// TIA Portal project "SIMULACION" (V16)

(* hardware
DEVICE "S7-1200 station_1"  S7-1200 Station
   slot 0: "Rack_0"  S7-1200 Rack  Rack  V1.0
   slot 1: "PLC_1"  CPU 1214C DC/DC/Rly  6ES7 214-1HG40-0XB0  V4.0
*)

// ===== PLC "PLC_1"  CPU 1214C DC/DC/Rly =====

VAR_GLOBAL   // PLC tag table "Default tag table"
   "ET0" AT %M0.0 : Bool;
   "ET1" AT %M0.1 : Bool;
   "ET2" AT %M0.2 : Bool;
   "ET3" AT %M0.3 : Bool;
   "ET4" AT %M0.4 : Bool;
   "ET5" AT %M0.5 : Bool;
   "ET6" AT %M0.6 : Bool;
   "ET7" AT %M0.7 : Bool;
   "ET8" AT %M1.0 : Bool;
   "ET9" AT %M1.1 : Bool;
   "ET10" AT %M1.2 : Bool;
   "ET11" AT %M1.3 : Bool;
   "ET12" AT %M1.4 : Bool;
   "ET13" AT %M1.5 : Bool;
   "ET14" AT %M1.6 : Bool;
   "ET15" AT %M1.7 : Bool;
   "ET16" AT %M2.0 : Bool;
   "ET17" AT %M2.1 : Bool;
   "ET18" AT %M2.2 : Bool;
   "MARCHA" AT %I0.0 : Bool;
   "TANQUEA" AT %Q0.0 : Bool;
   "TANQUEB" AT %Q0.1 : Bool;
   "W1" AT %Q0.2 : Bool;
   "W2" AT %Q0.3 : Bool;
   "W3" AT %Q0.4 : Bool;
   "W4" AT %Q0.5 : Bool;
   "W5" AT %Q0.6 : Bool;
END_VAR

// folder: System blocks/Program resources

DATA_BLOCK "TW1"   // DB2
{ S7_Optimized_Access := 'TRUE' }
AUTHOR : Simatic
FAMILY : IEC
NAME : IEC_TMR
VERSION : 1.0
// stored: InstanceOfName IEC_TIMER
"IEC_TIMER"
BEGIN
END_DATA_BLOCK

DATA_BLOCK "TW2"   // DB3
{ S7_Optimized_Access := 'TRUE' }
AUTHOR : Simatic
FAMILY : IEC
NAME : IEC_TMR
VERSION : 1.0
// stored: InstanceOfName IEC_TIMER
"IEC_TIMER"
BEGIN
END_DATA_BLOCK

DATA_BLOCK "TW3"   // DB4
{ S7_Optimized_Access := 'TRUE' }
AUTHOR : Simatic
FAMILY : IEC
NAME : IEC_TMR
VERSION : 1.0
// stored: InstanceOfName IEC_TIMER
"IEC_TIMER"
BEGIN
END_DATA_BLOCK

DATA_BLOCK "T4"   // DB5
{ S7_Optimized_Access := 'TRUE' }
AUTHOR : Simatic
FAMILY : IEC
NAME : IEC_TMR
VERSION : 1.0
// stored: InstanceOfName IEC_TIMER
"IEC_TIMER"
BEGIN
END_DATA_BLOCK

DATA_BLOCK "T5"   // DB6
{ S7_Optimized_Access := 'TRUE' }
AUTHOR : Simatic
FAMILY : IEC
NAME : IEC_TMR
VERSION : 1.0
// stored: InstanceOfName IEC_TIMER
"IEC_TIMER"
BEGIN
END_DATA_BLOCK

DATA_BLOCK "T6"   // DB7
{ S7_Optimized_Access := 'TRUE' }
AUTHOR : Simatic
FAMILY : IEC
NAME : IEC_TMR
VERSION : 1.0
// stored: InstanceOfName IEC_TIMER
"IEC_TIMER"
BEGIN
END_DATA_BLOCK

DATA_BLOCK "T7"   // DB8
{ S7_Optimized_Access := 'TRUE' }
AUTHOR : Simatic
FAMILY : IEC
NAME : IEC_TMR
VERSION : 1.0
// stored: InstanceOfName IEC_TIMER
"IEC_TIMER"
BEGIN
END_DATA_BLOCK

DATA_BLOCK "T8"   // DB9
{ S7_Optimized_Access := 'TRUE' }
AUTHOR : Simatic
FAMILY : IEC
NAME : IEC_TMR
VERSION : 1.0
// stored: InstanceOfName IEC_TIMER
"IEC_TIMER"
BEGIN
END_DATA_BLOCK

// folder: (top level)

ORGANIZATION_BLOCK "Main"   // OB1, LAD, ProgramCycle
TITLE = "Main Program Sweep (Cycle)"
{ S7_Optimized_Access := 'TRUE' }
VERSION : 0.1
BEGIN

REGION Network 1: Estado Inicial
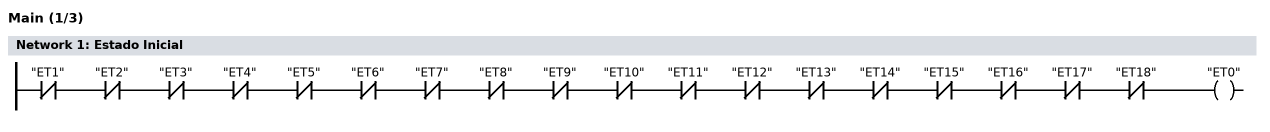
   RUNG wire#powerrail
      I_Contact( "ET1" )
      I_Contact( "ET2" )
      I_Contact( "ET3" )
      I_Contact( "ET4" )
      I_Contact( "ET5" )
      I_Contact( "ET6" )
      I_Contact( "ET7" )
      I_Contact( "ET8" )
      I_Contact( "ET9" )
      I_Contact( "ET10" )
      I_Contact( "ET11" )
      I_Contact( "ET12" )
      I_Contact( "ET13" )
      I_Contact( "ET14" )
      I_Contact( "ET15" )
      I_Contact( "ET16" )
      I_Contact( "ET17" )
      I_Contact( "ET18" )
      Coil( "ET0" )
   END_RUNG
   // the same network as SCL:
   "ET0" := NOT "ET1" AND NOT "ET2" AND NOT "ET3" AND NOT "ET4" AND NOT "ET5" AND NOT "ET6" AND NOT "ET7" AND NOT "ET8" AND NOT "ET9" AND NOT "ET10" AND NOT "ET11" AND NOT "ET12" AND NOT "ET13" AND NOT "ET14" AND NOT "ET15" AND NOT "ET16" AND NOT "ET17" AND NOT "ET18";
END_REGION

REGION Network 2: Etapas de transicion
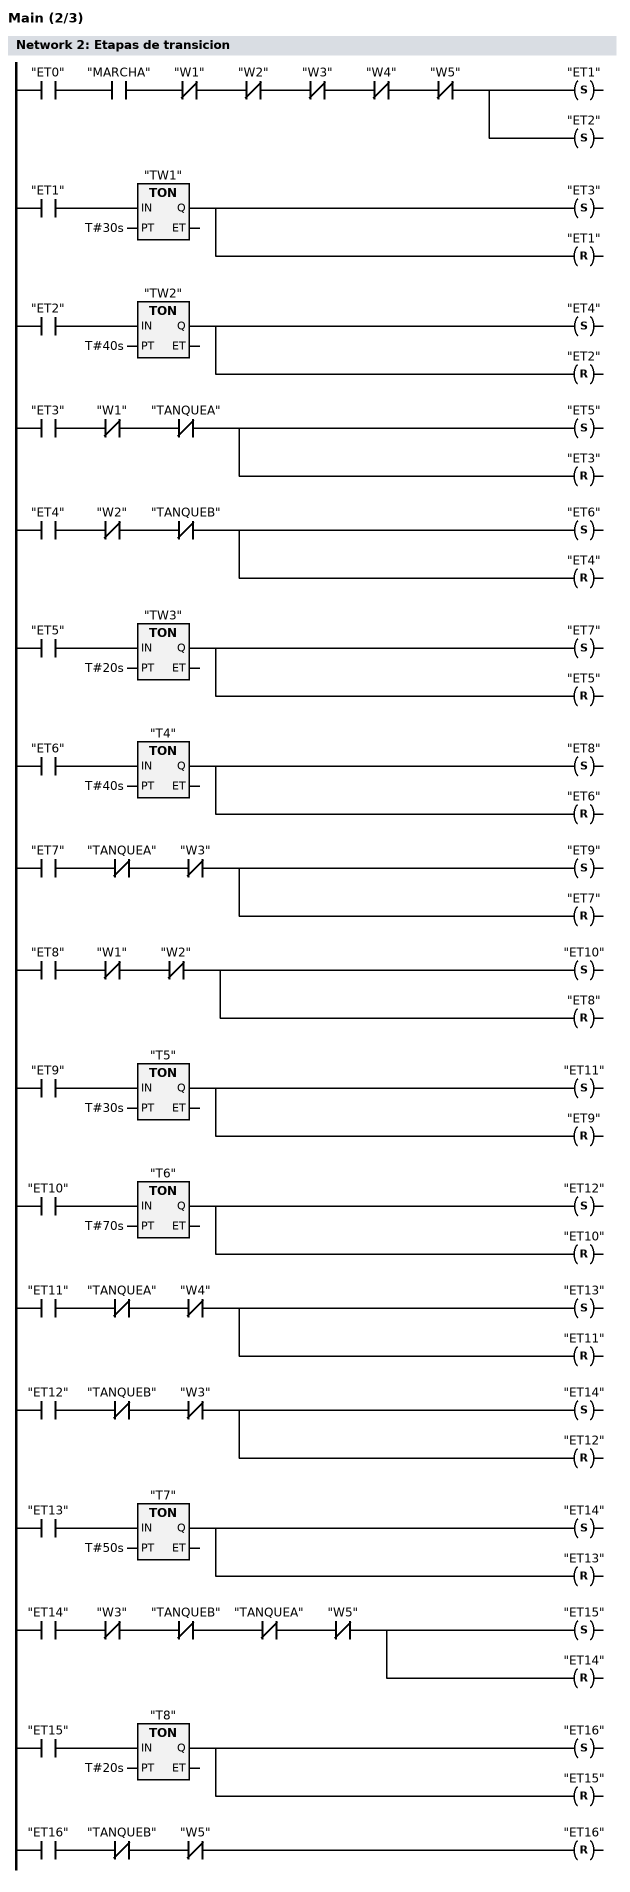
   IF "ET0" AND "MARCHA" AND NOT "W1" AND NOT "W2" AND NOT "W3" AND NOT "W4" AND NOT "W5" THEN
       "ET1" := TRUE;
       "ET2" := TRUE;
   END_IF;
   "TW1".TON(IN := "ET1", PT := T#30s);
   IF "TW1".Q THEN
       "ET3" := TRUE;
       "ET1" := FALSE;
   END_IF;
   "TW2".TON(IN := "ET2", PT := T#40s);
   IF "TW2".Q THEN
       "ET4" := TRUE;
       "ET2" := FALSE;
   END_IF;
   IF "ET3" AND NOT "W1" AND NOT "TANQUEA" THEN
       "ET5" := TRUE;
       "ET3" := FALSE;
   END_IF;
   IF "ET4" AND NOT "W2" AND NOT "TANQUEB" THEN
       "ET6" := TRUE;
       "ET4" := FALSE;
   END_IF;
   "TW3".TON(IN := "ET5", PT := T#20s);
   IF "TW3".Q THEN
       "ET7" := TRUE;
       "ET5" := FALSE;
   END_IF;
   "T4".TON(IN := "ET6", PT := T#40s);
   IF "T4".Q THEN
       "ET8" := TRUE;
       "ET6" := FALSE;
   END_IF;
   IF "ET7" AND NOT "TANQUEA" AND NOT "W3" THEN
       "ET9" := TRUE;
       "ET7" := FALSE;
   END_IF;
   IF "ET8" AND NOT "W1" AND NOT "W2" THEN
       "ET10" := TRUE;
       "ET8" := FALSE;
   END_IF;
   "T5".TON(IN := "ET9", PT := T#30s);
   IF "T5".Q THEN
       "ET11" := TRUE;
       "ET9" := FALSE;
   END_IF;
   "T6".TON(IN := "ET10", PT := T#70s);
   IF "T6".Q THEN
       "ET12" := TRUE;
       "ET10" := FALSE;
   END_IF;
   IF "ET11" AND NOT "TANQUEA" AND NOT "W4" THEN
       "ET13" := TRUE;
       "ET11" := FALSE;
   END_IF;
   IF "ET12" AND NOT "TANQUEB" AND NOT "W3" THEN
       "ET14" := TRUE;
       "ET12" := FALSE;
   END_IF;
   "T7".TON(IN := "ET13", PT := T#50s);
   IF "T7".Q THEN
       "ET14" := TRUE;
       "ET13" := FALSE;
   END_IF;
   IF "ET14" AND NOT "W3" AND NOT "TANQUEB" AND NOT "TANQUEA" AND NOT "W5" THEN
       "ET15" := TRUE;
       "ET14" := FALSE;
   END_IF;
   "T8".TON(IN := "ET15", PT := T#20s);
   IF "T8".Q THEN
       "ET16" := TRUE;
       "ET15" := FALSE;
   END_IF;
   IF "ET16" AND NOT "TANQUEB" AND NOT "W5" THEN "ET16" := FALSE; END_IF;
END_REGION

REGION Network 3: ETAPAS
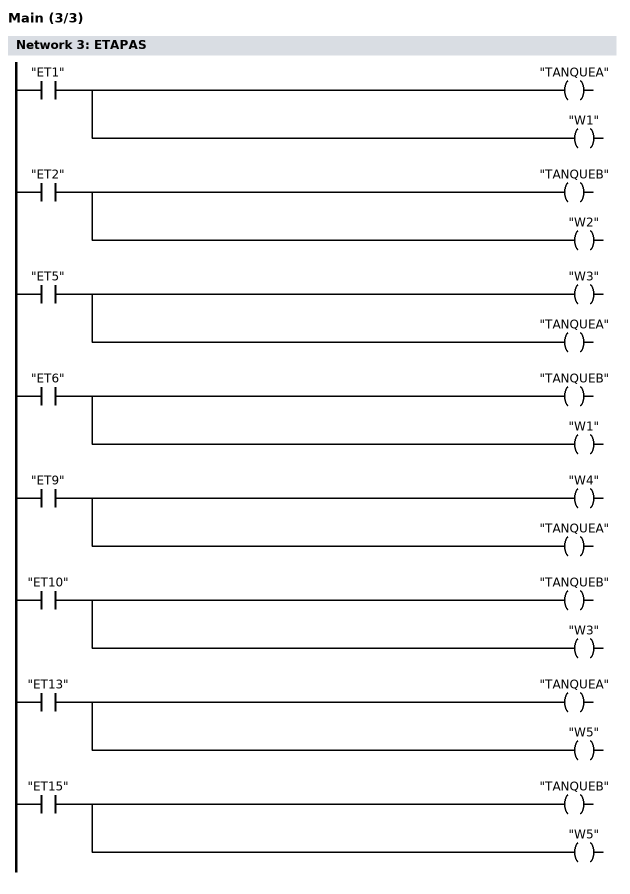
   RUNG wire#powerrail
      Contact( "ET1" )
      wire#w1
      Coil( "TANQUEA" )
   END_RUNG
   RUNG wire#w1
      Coil( "W1" )
   END_RUNG
   RUNG wire#powerrail
      Contact( "ET2" )
      wire#w2
      Coil( "TANQUEB" )
   END_RUNG
   RUNG wire#w2
      Coil( "W2" )
   END_RUNG
   RUNG wire#powerrail
      Contact( "ET5" )
      wire#w3
      Coil( "W3" )
   END_RUNG
   RUNG wire#w3
      Coil( "TANQUEA" )
   END_RUNG
   RUNG wire#powerrail
      Contact( "ET6" )
      wire#w4
      Coil( "TANQUEB" )
   END_RUNG
   RUNG wire#w4
      Coil( "W1" )
   END_RUNG
   RUNG wire#powerrail
      Contact( "ET9" )
      wire#w5
      Coil( "W4" )
   END_RUNG
   RUNG wire#w5
      Coil( "TANQUEA" )
   END_RUNG
   RUNG wire#powerrail
      Contact( "ET10" )
      wire#w6
      Coil( "TANQUEB" )
   END_RUNG
   RUNG wire#w6
      Coil( "W3" )
   END_RUNG
   RUNG wire#powerrail
      Contact( "ET13" )
      wire#w7
      Coil( "TANQUEA" )
   END_RUNG
   RUNG wire#w7
      Coil( "W5" )
   END_RUNG
   RUNG wire#powerrail
      Contact( "ET15" )
      wire#w8
      Coil( "TANQUEB" )
   END_RUNG
   RUNG wire#w8
      Coil( "W5" )
   END_RUNG
   // the same network as SCL:
   "TANQUEA" := "ET1";
   "W1" := "ET1";
   "TANQUEB" := "ET2";
   "W2" := "ET2";
   "W3" := "ET5";
   "TANQUEA" := "ET5";
   "TANQUEB" := "ET6";
   "W1" := "ET6";
   "W4" := "ET9";
   "TANQUEA" := "ET9";
   "TANQUEB" := "ET10";
   "W3" := "ET10";
   "TANQUEA" := "ET13";
   "W5" := "ET13";
   "TANQUEB" := "ET15";
   "W5" := "ET15";
END_REGION
END_ORGANIZATION_BLOCK